PROGRAM PRG2_Object_Detection
VAR
END_VAR

END_PROGRAM

(* stored: Version 1.1.0.1, ProductVersion 3.1.4024.12
   POU PRG2_Object_Detection: Id {e2c7d67f-cf17-4fff-92d2-d8b3d11a25b3}, SpecialFunc None *)
